SUBAPPLICATION AX_SwitchPic_2_1 (* Bild/ObjectPointer-Ziel umschalten VT; 2 Zustaende, Selector als AX-Adapter statt BOOL-InputVar (AX-Pendant zu MyLib::sys::SwitchPic_2_1) - schreibt bei jedem Update von DI1 das per DI1.D1 ausgewaehlte Ziel-Object-ID (pictures.down wenn TRUE, pictures.up wenn FALSE) auf den ObjectPointer Picture. *)
  (* Standard: 61499-2 *)
  (* Version 1.0, 2026-09-17, Franz Höpfinger, Meisterschulen am Ostbahnhof, Neu (Franz: 'dann Rectangle_Aktiv oder ID_NULL werfen auf ObjectPointer_Elevatorband_Ein ObjectPointer_Igelband_Ein ObjectPointer_Befuellband_Ein') - AX-Adapter-Pendant zu SwitchPic_2_1 (dort DI1:BOOL + externes EI-Event), hier DI1:AX-Socket dessen eigenes E1/D1 REQ/G direkt speist, kein externer Trigger noetig. *)
  PACKAGE MyLib::sys;
  IMPORT isobus::UT::Q::const::IDs::ID_NULL;
  IMPORT isobus::UT::Q::types::s2x1ObjectIDs;
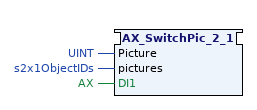
  VAR_INPUT
    Picture : UINT; (* Object ID of the ObjectPointer to write into *)
    pictures : isobus::UT::Q::types::s2x1ObjectIDs := (up := (u16ObjId := ID_NULL), down := (u16ObjId := ID_NULL)); (* die beiden Ziel-Object-IDs *)
  END_VAR
  SOCKETS
    DI1 : adapter::types::unidirectional::AX; (* Selector - down (pictures.down) wenn TRUE, up (pictures.up) wenn FALSE. Jedes Update schreibt sofort neu. *)
  END_SOCKETS
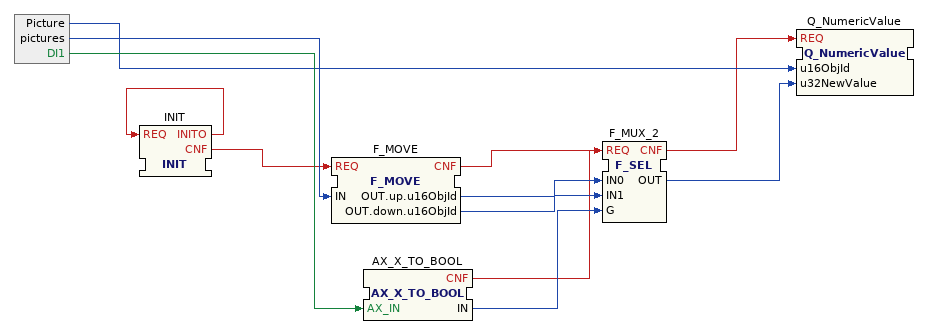
  FBS
    Q_NumericValue : isobus::UT::Q::Q_NumericValue;
    F_MOVE : iec61131::selection::F_MOVE; {SET_ATTRIBUTE(DataType, isobus::UT::Q::types::s2x1ObjectIDs)}
    F_MUX_2 : iec61131::selection::F_SEL;
    AX_X_TO_BOOL : adapter::conversion::unidirectional::AX_X_TO_BOOL;
    INIT : iec61131::booleanOperators::INIT;
  END_FBS
  EVENT_CONNECTIONS
    F_MUX_2.CNF TO Q_NumericValue.REQ;
    F_MOVE.CNF TO F_MUX_2.REQ;
    AX_X_TO_BOOL.CNF TO F_MUX_2.REQ;
    INIT.INITO TO INIT.REQ;
    INIT.CNF TO F_MOVE.REQ;
  END_CONNECTIONS
  DATA_CONNECTIONS
    Picture TO Q_NumericValue.u16ObjId;
    pictures TO F_MOVE.IN;
    F_MUX_2.OUT TO Q_NumericValue.u32NewValue;
    F_MOVE.OUT.up.u16ObjId TO F_MUX_2.IN0;
    F_MOVE.OUT.down.u16ObjId TO F_MUX_2.IN1;
    AX_X_TO_BOOL.IN TO F_MUX_2.G;
  END_CONNECTIONS
  ADAPTER_CONNECTIONS
    DI1 TO AX_X_TO_BOOL.AX_IN;
  END_CONNECTIONS
END_SUBAPPLICATION
